//==================================================================================================
//								RJM Maszyny sp. z o.o.
//									04.06.2022
//	Obsługa czujnika NC
// 	v1.0	|| TC v 3.1.4024.22		|| - pierwsza wersja
//==================================================================================================
FUNCTION_BLOCK FB_Czujnik_NC IMPLEMENTS ITF_Czujnik
VAR_INPUT
	bSymulacja								: BOOL;
END_VAR
VAR
	bWejscie						AT %I*	: BOOL;
END_VAR

//==================================================================================================
//								RJM Maszyny sp. z o.o.
//									04.06.2022
//	Obsługa czujnika  
// 	v1.0	|| TC v 3.1.4024.22		|| - pierwsza wersja
//==================================================================================================
PROPERTY CzyZadzialany : BOOL
GET
CzyZadzialany								:= NOT bWejscie;
END_GET
END_PROPERTY

END_FUNCTION_BLOCK

(* stored: Version 1.1.0.1, ProductVersion 3.1.4024.11
   POU FB_Czujnik_NC: Id {51ba7fa6-f7c0-4afd-bbfe-dc8f49c5646a}, SpecialFunc None
   Property CzyZadzialany: Id {fc66beb3-2c43-4161-beb6-70ba35ef7689}
   Get Get: Id {a9c273e3-8246-498a-9fbf-8e32a7aeaa7f} *)
